PROGRAM prg_OpenbaarToilet
VAR
	bSchakel1, bSchakel2, bSchakel3		AT		%I*		:BOOL;
	bLamp1, bLamp2, bLamp3				AT		%Q*		:BOOL;
	bVentilator							AT		%Q*		:BOOL;
	TimerOff: TOF;
END_VAR

bLamp1:= bSchakel1;
bLamp2:= bSchakel2;
bLamp3:= bSchakel3;
TimerOff(IN:= bSchakel1 OR bSchakel2 OR bSchakel3, PT:= T#5S, Q=> bVentilator);
//Dit werkt omdat de TOF op de FALLING EDGE detecteerd

END_PROGRAM

(* stored: Version 1.1.0.1, ProductVersion 3.1.4024.15
   POU prg_OpenbaarToilet: Id {764dfd20-4378-4478-a84a-d1d1d7df3ab5}, SpecialFunc None *)
